# EPICS IOC start-up script: iocsh/evm-mtca-init.iocsh
# .init.iocsh
# ===========

# ESS EVG command file for mrfioc2
# ================================

# PCIID address
mrmEvgSetupPCI($(DEV), $(PCIID))

dbLoadRecords("evm-mtca-300-ess.db", "SYS=$(IOC), D=$(DEV), EVG=$(DEV), FEVT=$(ESSEvtClockRate), FRF=$(ESSEvtClockRate), RFDIV=1")

var evrMrmTimeNSOverflowThreshold 100000

#EOF
